MOVL C01011 V=20 PL=LB000 ACC=LB001 DEC=LB001
MOVL C01012 V=20 PL=LB000 ACC=LB001 DEC=LB001
MOVL C01013 V=20 PL=LB000 ACC=LB001 DEC=LB001
MOVL C01014 V=25 PL=LB000 ACC=LB001 DEC=LB001
' rapid-dry
MOVL C01015 V=17 PL=LB000 ACC=LB001 DEC=LB001
MOVL C01016 V=25 PL=LB000 ACC=LB001 DEC=LB001
' bead-perimeter_outer
MOVL C01017 V=20 PL=LB000 ACC=LB001 DEC=LB001
MOVL C01018 V=20 PL=LB000 ACC=LB001 DEC=LB001
MOVL C01019 V=20 PL=LB000 ACC=LB001 DEC=LB001
MOVL C01020 V=20 PL=LB000 ACC=LB001 DEC=LB001
MOVL C01021 V=25 PL=LB000 ACC=LB001 DEC=LB001
' part 1 complete
' move to park position
MOVL C01022 V=17 PL=LB000 ACC=LB001 DEC=LB001
MOVL C01023 V=17 PL=LB000 ACC=LB001 DEC=LB001
' --------------------------------
' --------------------------------
' By Autodesk Fusion CAM 2.0.20494
' Tool = 1
' Spindle = 0 RPM
' Set Position Level
' Set Acceleration
' Program Start
' First Toolpath Point
END
